(* PLC project , 3S-Smart Software Solutions CODESYS Control Win *)

TYPE ModeEnum : (Off := 0, Auto := 1, Manual := 2);
END_TYPE

TYPE MotorConfig : STRUCT
  SpeedSetpoint : int := 1200;
  Enabled : bool := TRUE;
END_STRUCT;
END_TYPE

TYPE AlarmHistory : ARRAY[1..4] OF bool;
END_TYPE

TYPE DutyPercent : subrange;
END_TYPE

PROGRAM Main

PROGRAM Main
VAR
    Controller : MotorFb;
END_VAR
END_PROGRAM
END_PROGRAM

FUNCTION_BLOCK MotorFb

FUNCTION_BLOCK MotorFb
VAR_INPUT
    Enable : BOOL;
END_VAR
VAR
    Config : MotorConfig;
END_VAR
END_FUNCTION_BLOCK
END_FUNCTION_BLOCK

FUNCTION ComputeDuty

FUNCTION ComputeDuty : INT
ComputeDuty := 75;
END_FUNCTION
END_FUNCTION

CONFIGURATION PlantConfig
  RESOURCE CpuRes ON PLC
    TASK FastTask(INTERVAL := T#50ms, PRIORITY := 1);
    TASK SlowTask(INTERVAL := T#1000ms, PRIORITY := 5);
    PROGRAM MotorTaskInst : MotorFb;
  END_RESOURCE
END_CONFIGURATION
